TYPE PickerComRequest :
STRUCT
  Start : BOOL;
  Stop : BOOL;
  GoHome : BOOL;
  Halt : BOOL;
END_STRUCT
END_TYPE

(* stored: Version 1.1.0.1
   DUT PickerComRequest: Id {cec60d3d-7d51-46ef-824f-5b605d126f44} *)
